PROGRAM MAIN
VAR;
	InitEnOcean: EnOCean;
	Switches: SwitchEnOcean;
	Search: SearchEnOcean;
END_VAR

InitEnOcean();
Switches();
Search();

END_PROGRAM

(* stored: Version 1.1.0.1, ProductVersion 3.1.4022.16
   POU MAIN: Id {0968eccf-1f42-4a9c-9ff8-6dadd354813e}, SpecialFunc None *)
